// TIA Portal V19 export
TYPE "lexchangetray_typeroller_signalTM_Monitor"
// Type: Bool
// stored: Access Published
   STRUCT
      trayAutomaticDischargeDetectionEm1 : Bool;
      trayAutomaticFeedingDetectionEm1 : Bool;
      restraintTrayAntiReverseDetection2Em1 : Bool;
      restraintTrayAntiReverseDetection1Em1 : Bool;
      simulationed : Bool;
   END_STRUCT;
END_TYPE
